(* IEC 61131-3 sources: Hearthline/project/control/programs/body-preparation, 1 file *)

(* ---- area-01-vplc-01.st ---- *)
PROGRAM BodyPreparationBatch
VAR_INPUT
    StartBatch : BOOL;
    SafetyReady : BOOL;
    ResetBatch : BOOL;
    TripActive : BOOL;
    BatchMass : REAL;
    WaterFlow : REAL;
    MixerLevel : REAL;
    MixerTemperature : REAL;
    MixingEnergy : REAL;
    SlipDensity : REAL;
    SlipViscosity : REAL;
    SlipTemperature : REAL;
    ConditioningLevel : REAL;
    TransferFlow : REAL;
END_VAR
VAR_OUTPUT
    PhaseCode : DINT;
    WaterValveCommand : INT;
    SilicatePumpCommand : INT;
    BallClayFeederCommand : INT;
    KaolinFeederCommand : INT;
    FeldsparFeederCommand : INT;
    QuartzFeederCommand : INT;
    MixerCommand : INT;
    ScreenCommand : INT;
    MagnetCommand : INT;
    ConditioningAgitatorCommand : INT;
    HeaterCommand : INT;
    TransferValveCommand : INT;
    TransferPumpCommand : INT;
END_VAR
VAR
    Step : DINT := 0;
    StepTimer : TON;
END_VAR

CASE Step OF
0:
    PhaseCode := 0;
    WaterValveCommand := 0;
    SilicatePumpCommand := 0;
    BallClayFeederCommand := 0;
    KaolinFeederCommand := 0;
    FeldsparFeederCommand := 0;
    QuartzFeederCommand := 0;
    MixerCommand := 0;
    ScreenCommand := 0;
    MagnetCommand := 1;
    ConditioningAgitatorCommand := 0;
    HeaterCommand := 0;
    TransferValveCommand := 0;
    TransferPumpCommand := 0;
    IF StartBatch AND SafetyReady THEN Step := 10; END_IF;
10:
    PhaseCode := 10;
    WaterValveCommand := 1;
    SilicatePumpCommand := 0;
    BallClayFeederCommand := 0;
    KaolinFeederCommand := 0;
    FeldsparFeederCommand := 0;
    QuartzFeederCommand := 0;
    MixerCommand := 0;
    ScreenCommand := 0;
    MagnetCommand := 1;
    ConditioningAgitatorCommand := 0;
    HeaterCommand := 0;
    TransferValveCommand := 0;
    TransferPumpCommand := 0;
    StepTimer(IN := TRUE, PT := T#600ms);
    IF StepTimer.Q THEN Step := 20; END_IF;
20:
    PhaseCode := 20;
    WaterValveCommand := 0;
    SilicatePumpCommand := 1;
    BallClayFeederCommand := 0;
    KaolinFeederCommand := 0;
    FeldsparFeederCommand := 0;
    QuartzFeederCommand := 0;
    MixerCommand := 0;
    ScreenCommand := 0;
    MagnetCommand := 1;
    ConditioningAgitatorCommand := 0;
    HeaterCommand := 0;
    TransferValveCommand := 0;
    TransferPumpCommand := 0;
    StepTimer(IN := TRUE, PT := T#250ms);
    IF StepTimer.Q THEN Step := 30; END_IF;
30:
    PhaseCode := 30;
    WaterValveCommand := 0;
    SilicatePumpCommand := 0;
    BallClayFeederCommand := 1;
    KaolinFeederCommand := 0;
    FeldsparFeederCommand := 0;
    QuartzFeederCommand := 0;
    MixerCommand := 0;
    ScreenCommand := 0;
    MagnetCommand := 1;
    ConditioningAgitatorCommand := 0;
    HeaterCommand := 0;
    TransferValveCommand := 0;
    TransferPumpCommand := 0;
    StepTimer(IN := TRUE, PT := T#600ms);
    IF StepTimer.Q THEN Step := 40; END_IF;
40:
    PhaseCode := 40;
    WaterValveCommand := 0;
    SilicatePumpCommand := 0;
    BallClayFeederCommand := 0;
    KaolinFeederCommand := 1;
    FeldsparFeederCommand := 0;
    QuartzFeederCommand := 0;
    MixerCommand := 0;
    ScreenCommand := 0;
    MagnetCommand := 1;
    ConditioningAgitatorCommand := 0;
    HeaterCommand := 0;
    TransferValveCommand := 0;
    TransferPumpCommand := 0;
    StepTimer(IN := TRUE, PT := T#600ms);
    IF StepTimer.Q THEN Step := 50; END_IF;
50:
    PhaseCode := 50;
    WaterValveCommand := 0;
    SilicatePumpCommand := 0;
    BallClayFeederCommand := 0;
    KaolinFeederCommand := 0;
    FeldsparFeederCommand := 1;
    QuartzFeederCommand := 0;
    MixerCommand := 0;
    ScreenCommand := 0;
    MagnetCommand := 1;
    ConditioningAgitatorCommand := 0;
    HeaterCommand := 0;
    TransferValveCommand := 0;
    TransferPumpCommand := 0;
    StepTimer(IN := TRUE, PT := T#400ms);
    IF StepTimer.Q THEN Step := 60; END_IF;
60:
    PhaseCode := 60;
    WaterValveCommand := 0;
    SilicatePumpCommand := 0;
    BallClayFeederCommand := 0;
    KaolinFeederCommand := 0;
    FeldsparFeederCommand := 0;
    QuartzFeederCommand := 1;
    MixerCommand := 0;
    ScreenCommand := 0;
    MagnetCommand := 1;
    ConditioningAgitatorCommand := 0;
    HeaterCommand := 0;
    TransferValveCommand := 0;
    TransferPumpCommand := 0;
    StepTimer(IN := TRUE, PT := T#400ms);
    IF StepTimer.Q THEN Step := 70; END_IF;
70:
    PhaseCode := 70;
    WaterValveCommand := 0;
    SilicatePumpCommand := 0;
    BallClayFeederCommand := 0;
    KaolinFeederCommand := 0;
    FeldsparFeederCommand := 0;
    QuartzFeederCommand := 0;
    MixerCommand := 1;
    ScreenCommand := 0;
    MagnetCommand := 1;
    ConditioningAgitatorCommand := 0;
    HeaterCommand := 0;
    TransferValveCommand := 0;
    TransferPumpCommand := 0;
    StepTimer(IN := TRUE, PT := T#6000ms);
    IF StepTimer.Q THEN Step := 80; END_IF;
80:
    PhaseCode := 80;
    WaterValveCommand := 0;
    SilicatePumpCommand := 0;
    BallClayFeederCommand := 0;
    KaolinFeederCommand := 0;
    FeldsparFeederCommand := 0;
    QuartzFeederCommand := 0;
    MixerCommand := 0;
    ScreenCommand := 1;
    MagnetCommand := 1;
    ConditioningAgitatorCommand := 0;
    HeaterCommand := 0;
    TransferValveCommand := 0;
    TransferPumpCommand := 0;
    StepTimer(IN := TRUE, PT := T#750ms);
    IF StepTimer.Q THEN Step := 90; END_IF;
90:
    PhaseCode := 90;
    WaterValveCommand := 0;
    SilicatePumpCommand := 0;
    BallClayFeederCommand := 0;
    KaolinFeederCommand := 0;
    FeldsparFeederCommand := 0;
    QuartzFeederCommand := 0;
    MixerCommand := 0;
    ScreenCommand := 0;
    MagnetCommand := 2;
    ConditioningAgitatorCommand := 0;
    HeaterCommand := 0;
    TransferValveCommand := 0;
    TransferPumpCommand := 0;
    StepTimer(IN := TRUE, PT := T#250ms);
    IF StepTimer.Q THEN Step := 100; END_IF;
100:
    PhaseCode := 100;
    WaterValveCommand := 0;
    SilicatePumpCommand := 0;
    BallClayFeederCommand := 0;
    KaolinFeederCommand := 0;
    FeldsparFeederCommand := 0;
    QuartzFeederCommand := 0;
    MixerCommand := 0;
    ScreenCommand := 0;
    MagnetCommand := 1;
    ConditioningAgitatorCommand := 1;
    HeaterCommand := 0;
    TransferValveCommand := 0;
    TransferPumpCommand := 0;
    StepTimer(IN := TRUE, PT := T#24000ms);
    IF StepTimer.Q THEN Step := 110; END_IF;
110:
    PhaseCode := 110;
    WaterValveCommand := 0;
    SilicatePumpCommand := 0;
    BallClayFeederCommand := 0;
    KaolinFeederCommand := 0;
    FeldsparFeederCommand := 0;
    QuartzFeederCommand := 0;
    MixerCommand := 0;
    ScreenCommand := 0;
    MagnetCommand := 1;
    ConditioningAgitatorCommand := 1;
    HeaterCommand := 0;
    TransferValveCommand := 0;
    TransferPumpCommand := 0;
    StepTimer(IN := TRUE, PT := T#500ms);
    IF StepTimer.Q THEN Step := 120; END_IF;
120:
    PhaseCode := 120;
    WaterValveCommand := 0;
    SilicatePumpCommand := 0;
    BallClayFeederCommand := 0;
    KaolinFeederCommand := 0;
    FeldsparFeederCommand := 0;
    QuartzFeederCommand := 0;
    MixerCommand := 0;
    ScreenCommand := 0;
    MagnetCommand := 1;
    ConditioningAgitatorCommand := 1;
    HeaterCommand := 1;
    TransferValveCommand := 0;
    TransferPumpCommand := 0;
    StepTimer(IN := TRUE, PT := T#1500ms);
    IF StepTimer.Q THEN Step := 130; END_IF;
130:
    PhaseCode := 130;
    WaterValveCommand := 0;
    SilicatePumpCommand := 0;
    BallClayFeederCommand := 0;
    KaolinFeederCommand := 0;
    FeldsparFeederCommand := 0;
    QuartzFeederCommand := 0;
    MixerCommand := 0;
    ScreenCommand := 0;
    MagnetCommand := 1;
    ConditioningAgitatorCommand := 1;
    HeaterCommand := 0;
    TransferValveCommand := 1;
    TransferPumpCommand := 1;
    StepTimer(IN := TRUE, PT := T#1250ms);
    IF StepTimer.Q THEN Step := 140; END_IF;
140:
    PhaseCode := 140;
    WaterValveCommand := 0;
    SilicatePumpCommand := 0;
    BallClayFeederCommand := 0;
    KaolinFeederCommand := 0;
    FeldsparFeederCommand := 0;
    QuartzFeederCommand := 0;
    MixerCommand := 0;
    ScreenCommand := 0;
    MagnetCommand := 1;
    ConditioningAgitatorCommand := 0;
    HeaterCommand := 0;
    TransferValveCommand := 0;
    TransferPumpCommand := 0;
    StepTimer(IN := TRUE, PT := T#250ms);
    IF StepTimer.Q THEN Step := 0; END_IF;
900:
    PhaseCode := 900;
    WaterValveCommand := 0;
    SilicatePumpCommand := 0;
    BallClayFeederCommand := 0;
    KaolinFeederCommand := 0;
    FeldsparFeederCommand := 0;
    QuartzFeederCommand := 0;
    MixerCommand := 0;
    ScreenCommand := 0;
    MagnetCommand := 1;
    ConditioningAgitatorCommand := 0;
    HeaterCommand := 0;
    TransferValveCommand := 0;
    TransferPumpCommand := 0;
    IF ResetBatch AND SafetyReady AND NOT TripActive THEN Step := 0; END_IF;
END_CASE;
END_PROGRAM
